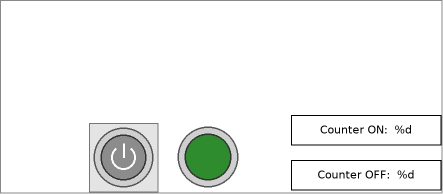
VISUALIZATION Visu_Lamp  // 443x194
    Lamp1 (173,122 70x70), variable: MAIN.fbUmlSc_Lamp.ObLamp, style: Lamp-Lamp1-Green
    PowerSwitch (69,123 109x69), variable: MAIN.fbUmlSc_Lamp.bPower, behaviour: TOGGLE, style: Switch-PowerSwitch-Gray
    Rectangle (291,115 150x30), "Counter ON: %d", text variable: MAIN.fbUmlSc_Lamp.nCounterOn
    Rectangle (291,160 150x30), "Counter OFF: %d", text variable: MAIN.fbUmlSc_Lamp.nCounterOff
END_VISUALIZATION

(* stored: Version 1.1.0.1
   Visu Visu_Lamp: Id {089ba7ce-990f-4333-a285-051a593f54ee} *)
